PROGRAM MAIN
VAR

END_VAR

POU_Example();

END_PROGRAM

(* stored: Version 1.1.0.1, ProductVersion 3.1.4022.12
   POU MAIN: Id {984fee79-3eda-4ea9-b09e-d08ce056b358}, SpecialFunc None *)
